// ---- tc_mca_std_lib/VISUs/PneumaticsVisu.TcVIS
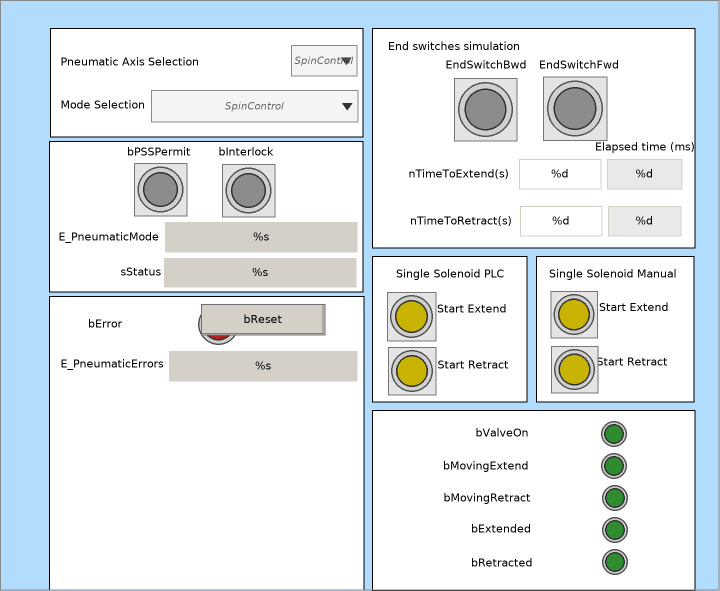
VISUALIZATION PneumaticsVisu  // 720x591
    Rectangle (50,28 313x109)
    Label (55,47 150x30), "Pneumatic Axis Selection"
    Rectangle (372,28 323x220)
    Label (379,30 150x33), "End switches simulation"
    Label (411,50 150x30), "EndSwitchBwd"
    SpinControl (291,45 66x31), variable: MAIN.hmiPneumaticAxisSelection
        p651134158: GVL_APP.nPNEUMATIC_AXIS_NUM
    Label (504,50 150x30), "EndSwitchFwd"
    Rectangle (49,296 315x294)
    Textfield (519,159 82x30), "%d", text variable: MAIN.afbPneumaticAxes[MAIN.hmiPneumaticAxisSelection].stPneumaticAxisStruct.stPneumaticAxisConfig.nTimeToExtend
        OnMouseClick: write MAIN.afbPneumaticAxes[MAIN.hmiPneumaticAxisSelection].stPneumaticAxisStruct.stPneumaticAxisConfig.nTimeToExtend via Default
    Label (384,159 150x30), "nTimeToExtend(s)"
    Label (386,206 150x30), "nTimeToRetract(s)"
    Label (28,90 150x30), "Mode Selection"
    Rectangle (49,141 314x151)
    Label (30,309 150x30), "bError"
    Lamp1 (126,301 185x47), variable: MAIN.afbPneumaticAxes[MAIN.hmiPneumaticAxisSelection].stPneumaticAxisStruct.stPneumaticAxisStatus.bError, style: Lamp-Lamp1-Red
    Label (37,349 150x30), "E_PneumaticErrors"
    Textfield (169,351 188x30), "%s", text variable: MAIN.afbPneumaticAxes[MAIN.hmiPneumaticAxisSelection].stPneumaticAxisStruct.ePneumaticAxisErrors, text list: 'languageSupport'
    Rectangle (372,256 155x146)
    Rectangle (536,256 158x146)
    Rectangle (372,410 323x181)
    Label (538,259 150x30), "Single Solenoid Manual"
    PushSwitchLed (549,291 50x47), variable: MAIN.afbPneumaticAxes[MAIN.hmiPneumaticAxisSelection].stPneumaticAxisStruct.stPneumaticAxisInputs.bOpenManual, behaviour: TOGGLE, style: Switch-PushSwitchLed-Yellow
    Label (592,293 84x29), "Start Extend"
    Label (557,347 150x30), "Start Retract"
    Label (375,259 150x30), "Single Solenoid PLC"
    PushSwitchLed (387,292 49x49), variable: MAIN.afbPneumaticAxes[MAIN.hmiPneumaticAxisSelection].stPneumaticAxisStruct.stPneumaticAxisControl.bExtend, behaviour: TOGGLE, style: Switch-PushSwitchLed-Yellow
    PushSwitchLed (388,347 48x48), variable: MAIN.afbPneumaticAxes[MAIN.hmiPneumaticAxisSelection].stPneumaticAxisStruct.stPneumaticAxisControl.bRetract, behaviour: TOGGLE, style: Switch-PushSwitchLed-Yellow
    Label (427,418 150x30), "bValveOn"
    Lamp1 (539,419 150x30), variable: MAIN.afbPneumaticAxes[MAIN.hmiPneumaticAxisSelection].stPneumaticAxisStruct.stPneumaticAxisOutputs.bValveOn, style: Lamp-Lamp1-Green
    Label (411,451 150x30), "bMovingExtend"
    Lamp1 (539,451 150x30), variable: MAIN.afbPneumaticAxes[MAIN.hmiPneumaticAxisSelection].stPneumaticAxisStruct.stPneumaticAxisStatus.bExtending, style: Lamp-Lamp1-Green
    Lamp1 (540,483 150x30), variable: MAIN.afbPneumaticAxes[MAIN.hmiPneumaticAxisSelection].stPneumaticAxisStruct.stPneumaticAxisStatus.bRetracting, style: Lamp-Lamp1-Green
    Lamp1 (540,515 150x30), variable: MAIN.afbPneumaticAxes[MAIN.hmiPneumaticAxisSelection].stPneumaticAxisStruct.stPneumaticAxisStatus.bExtended, style: Lamp-Lamp1-Green
    Lamp1 (540,547 150x30), variable: MAIN.afbPneumaticAxes[MAIN.hmiPneumaticAxisSelection].stPneumaticAxisStruct.stPneumaticAxisStatus.bRetracted, style: Lamp-Lamp1-Green
    Label (412,483 150x30), "bMovingRetract"
    Label (426,514 150x30), "bExtended"
    Label (397,294 150x30), "Start Extend"
    Label (398,350 150x30), "Start Retract"
    Label (427,548 150x30), "bRetracted"
    Button (201,304 124x31), "bReset"
        toggle MAIN.afbPneumaticAxes[MAIN.hmiPneumaticAxisSelection].stPneumaticAxisStruct.stPneumaticAxisControl.bReset
    PushSwitchLed (549,346 51x47), variable: MAIN.afbPneumaticAxes[MAIN.hmiPneumaticAxisSelection].stPneumaticAxisStruct.stPneumaticAxisInputs.bCloseManual, behaviour: TOGGLE, style: Switch-PushSwitchLed-Yellow
    Label (84,137 150x30), "bPSSPermit"
    Label (34,222 150x30), "E_PneumaticMode"
    Textfield (165,222 192x30), "%s", text variable: MAIN.afbPneumaticAxes[MAIN.hmiPneumaticAxisSelection].stPneumaticAxisStruct.ePneumaticAxisMode, text list: 'languageSupport'
    Textfield (164,258 192x29), "%s", text variable: MAIN.afbPneumaticAxes[MAIN.hmiPneumaticAxisSelection].stPneumaticAxisStruct.stPneumaticAxisStatus.sStatus, text list: 'languageSupport'
    Label (66,257 150x30), "sStatus"
    Textfield (520,206 82x30), "%d", text variable: MAIN.afbPneumaticAxes[MAIN.hmiPneumaticAxisSelection].stPneumaticAxisStruct.stPneumaticAxisConfig.nTimeToRetract
        OnMouseClick: write MAIN.afbPneumaticAxes[MAIN.hmiPneumaticAxisSelection].stPneumaticAxisStruct.stPneumaticAxisConfig.nTimeToRetract via Default
    Textfield (607,159 75x30), "%d", text variable: MAIN.afbPneumaticAxes[MAIN.hmiPneumaticAxisSelection].fbTimerExtend.ET
    Textfield (608,206 73x30), "%d", text variable: MAIN.afbPneumaticAxes[MAIN.hmiPneumaticAxisSelection].fbTimerRetract.ET
    SpinControl (151,90 207x32), variable: MAIN.afbPneumaticAxes[MAIN.hmiPneumaticAxisSelection].stPneumaticAxisStruct.ePneumaticAxisMode
    Label (570,132 150x30), "Elapsed time (ms)"
    PushSwitchLed (454,77 63x65), variable: MAIN.afbPneumaticAxes[MAIN.hmiPneumaticAxisSelection].stPneumaticAxisStruct.stPneumaticAxisInputs.bEndSwitchBwd, behaviour: TOGGLE, style: Switch-PushSwitchLed-Gray
    PushSwitchLed (543,76 64x65), variable: MAIN.afbPneumaticAxes[MAIN.hmiPneumaticAxisSelection].stPneumaticAxisStruct.stPneumaticAxisInputs.bEndSwitchFwd, behaviour: TOGGLE, style: Switch-PushSwitchLed-Gray
    PushSwitchLed (134,163 53x53), variable: MAIN.afbPneumaticAxes[MAIN.hmiPneumaticAxisSelection].stPneumaticAxisStruct.stPneumaticAxisInputs.bPSSPermit, behaviour: TOGGLE, style: Switch-PushSwitchLed-Gray
    PushSwitchLed (222,164 53x53), variable: MAIN.afbPneumaticAxes[MAIN.hmiPneumaticAxisSelection].stPneumaticAxisStruct.stPneumaticAxisControl.bInterlock, behaviour: TOGGLE, style: Switch-PushSwitchLed-Gray
    Label (171,137 150x30), "bInterlock"
END_VISUALIZATION

// ---- tc_mca_std_lib/VISUs_Org/languageSupport_1.TcTLO
TEXTLIST languageSupport_1
  axesAvailable = 'PLC Axes available: %d' | Test: 'Alt language'
  velocity = 'Velocity:'
  actposition = 'Actual Position:'
  enable = 'Enable Axis'
  enFW = 'Fwd Enable'
  enBW = 'Bwd Enable'
  axisSel = 'Axis Selected:'
  actVelocity = 'Actual Velocity:'
  errID = 'Error ID:'
  bEnabled = 'Axis Enabled'
  bCommandAborted = 'Command Aborted'
  bBusy = 'Busy'
  bDone = 'Command Done'
  bResetDone = 'Reset Complete'
  bHomed = 'Calibrated'
  bFwEnabled = 'Fwd movement enabled'
  bBwEnabled = 'Bwd movement enabled'
  bError = 'Error'
  fVelocity = 'Target Velocity:'
  fAcceleration = 'Target Accel.:'
  fDeceleration = 'Target Decel.:'
  fPosition = 'Target Position:'
  moveAbsolute = 'Absolute position move'
  toggle = 'Toggle'
  moveVelocity = 'Constant velocity move'
  bExecute = 'Motion function executed'
  moveRelative = 'Relative position move'
  moveModulo = 'Modulo position move'
  reset = 'Reset axis'
  stop = 'Stop motion'
  jogBw = 'Jog Backward'
  jogFw = 'Jog Forward'
  bGeared = 'In Gear'
  masterGear = 'Master Axis'
  gearRatio = 'Gear Ratio'
  gearIn = 'Gear In'
  gearOut = 'Gear Out'
  eHomeToLimit_Bwd = 'Bwd Limit'
  eHomeToLimit_Fwd = 'Fwd Limit'
  eHomeToRef_Bwd = 'Home Switch Bwd '
  eHomeToRef_Fwd = 'Home Switch Fwd '
  eHomeToEncPulse_Bwd = 'Enc Pulse Bwd '
  eHomeToEncPulse_Fwd = 'Enc Pulse Fwd'
  eHomeToEncPulse_viaBwdLimit = 'Enc Pulse via Bwd Limit'
  eHomeToEncPulse_viaFwdLimit = 'Enc Pulse via Fwd Limit'
  eHomeToBlock_Bwd = 'Home To Block Bwd Lag Based'
  eHomeToBlock_Fwd = 'Home To Block Fwd Lag Based'
  eHomeDirect = 'Home Direct'
  fHomePosition = 'Set Pos after Homing'
  fHomeFinishDistance = 'Relative Move after Homing'
  halt = 'Halt Motion'
  bInterlockBwd = 'Interlock Bwd'
  bInterlockFwd = 'Interlock Fwd'
  Home = 'HOME'
  eWriteParameter = 'Write Parameter'
  eReadParameter = 'Read Parameter'
  fWriteAxisParameter = 'Parameter to write'
  fReadAxisParameter = 'Parameter'
  bLocalMode = 'Local Mode'
  bInVelocity = 'Target Velocity reached'
   = ''
END_TEXTLIST

// ---- tc_mca_std_lib/VISUs_Org/MainVisu_1.TcVIS
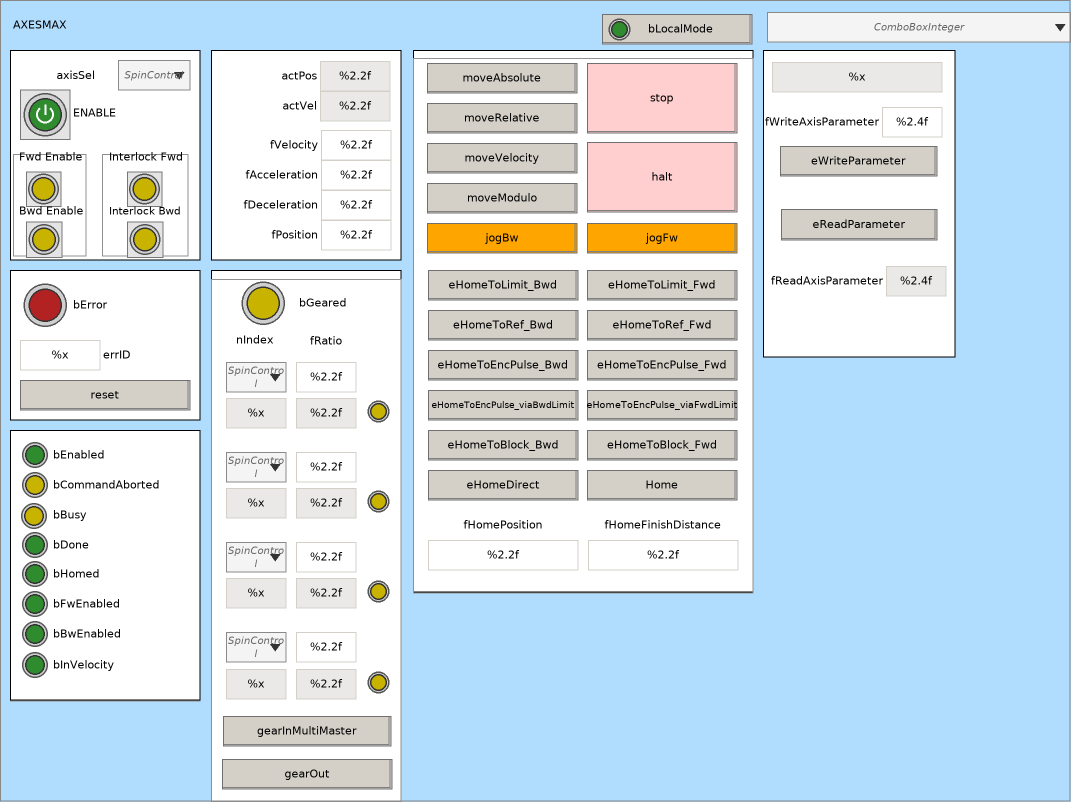
VISUALIZATION MainVisu_1  // 1071x802
    Rectangle (413,50 340x542)
    GroupBox (413,50 340x543)
        Button (174,92 150x70), "halt", pressed state: GVL.astAxes[Main.hmiAxisSelection].stControl.bHalt, input disabled if: GVL.astAxes[MAIN.hmiAxisSelection].stStatus.bGeared, text list: "languageSupport", text index: "halt"
            toggle GVL.astAxes[Main.hmiAxisSelection].stControl.bHalt
        Button (174,420 150x30), "Home", input disabled if: GVL.astAxes[MAIN.hmiAxisSelection].stStatus.bGeared, text list: 'languageSupport', text index: "Home"
            OnMouseClick: execute { GVL.astAxes[Main.hmiAxisSelection].stControl.eCommand:=E_MotionFunctions.eHome; GVL.astAxes[Main.hmiAxisSelection].stControl.bExecute:=TRUE; }
        Button (15,380 150x30), "eHomeToBlock_Bwd", input disabled if: GVL.astAxes[MAIN.hmiAxisSelection].stStatus.bGeared, text list: 'languageSupport', text index: "eHomeToBlock_Bwd"
            OnMouseClick: execute {
                GVL.astAxes[Main.hmiAxisSelection].stControl.eCommand:=E_MotionFunctions.eHome;
                GVL.astAxes[Main.hmiAxisSelection].stConfig.eHomeSeq:=E_HomingRoutines.eHomeToBlock_Bwd;
                GVL.astAxes[Main.hmiAxisSelection].stControl.bExecute:=TRUE;
            }
    Rectangle (211,270 190x531)
    GroupBox (211,271 190x531)
        SpinControl (15,91 60x30), variable: GVL.astAxes[MAIN.hmiAxisSelection].stConfig.astMultiMasterAxis[1].nIndex
            p651134158: GVL_APP.nAXIS_NUM
        Textfield (85,91 60x30), "%2.2f", text variable: GVL.astAxes[MAIN.hmiAxisSelection].stConfig.astMultiMasterAxis[1].fRatio
            OnMouseClick: write the text variable via Default
        Textfield (80,55 70x30), "fRatio", text list: "languageSupport", text index: "gearRatio"
        Button (12,445 168x30), "gearInMultiMaster", text list: "languageSupport", text index: "gearIn"
            OnMouseClick: execute { GVL.astAxes[Main.hmiAxisSelection].stControl.eCommand:=E_MotionFunctions.eGearInMultiMaster; GVL.astAxes[Main.hmiAxisSelection].stControl.bExecute:=TRUE; }
        SpinControl (15,181 60x30), variable: GVL.astAxes[MAIN.hmiAxisSelection].stConfig.astMultiMasterAxis[2].nIndex
            p651134158: GVL_APP.nAXIS_NUM
        SpinControl (15,271 60x30), variable: GVL.astAxes[MAIN.hmiAxisSelection].stConfig.astMultiMasterAxis[3].nIndex
            p651134158: GVL_APP.nAXIS_NUM
        SpinControl (15,361 60x30), variable: GVL.astAxes[MAIN.hmiAxisSelection].stConfig.astMultiMasterAxis[4].nIndex
            p651134158: GVL_APP.nAXIS_NUM
        Textfield (85,181 60x30), "%2.2f", text variable: GVL.astAxes[MAIN.hmiAxisSelection].stConfig.astMultiMasterAxis[2].fRatio
            OnMouseClick: write the text variable via Default
        Textfield (85,271 60x30), "%2.2f", text variable: GVL.astAxes[MAIN.hmiAxisSelection].stConfig.astMultiMasterAxis[3].fRatio
            OnMouseClick: write the text variable via Default
        Textfield (85,361 60x30), "%2.2f", text variable: GVL.astAxes[MAIN.hmiAxisSelection].stConfig.astMultiMasterAxis[4].fRatio
            OnMouseClick: write the text variable via Default
        Button (11,488 170x30), "gearOut", text list: "languageSupport", text index: "gearOut"
            OnMouseClick: execute { GVL.astAxes[Main.hmiAxisSelection].stControl.eCommand:=E_MotionFunctions.eGearOut; GVL.astAxes[Main.hmiAxisSelection].stControl.bExecute:=TRUE; }
        Textfield (9,54 70x30), "nIndex", text list: "languageSupport", text index: "masterGear"
        Textfield (85,127 60x30), "%2.2f", text variable: GVL.astAxes[MAIN.hmiAxisSelection].Axis.PlcToNc.GearRatio1
        Textfield (15,127 60x30), "%x", text variable: GVL.astAxes[MAIN.hmiAxisSelection].stConfig.astMultiMasterAxisLatched[1].nIndex
        Textfield (85,217 60x30), "%2.2f", text variable: GVL.astAxes[MAIN.hmiAxisSelection].Axis.PlcToNc.GearRatio2
        Textfield (15,217 60x30), "%x", text variable: GVL.astAxes[MAIN.hmiAxisSelection].stConfig.astMultiMasterAxisLatched[2].nIndex
        Textfield (85,307 60x30), "%2.2f", text variable: GVL.astAxes[MAIN.hmiAxisSelection].Axis.PlcToNc.GearRatio3
        Textfield (15,307 60x30), "%x", text variable: GVL.astAxes[MAIN.hmiAxisSelection].stConfig.astMultiMasterAxisLatched[3].nIndex
        Textfield (85,398 60x30), "%2.2f", text variable: GVL.astAxes[MAIN.hmiAxisSelection].Axis.PlcToNc.GearRatio4
        Textfield (15,398 60x30), "%x", text variable: GVL.astAxes[MAIN.hmiAxisSelection].stConfig.astMultiMasterAxisLatched[4].nIndex
        Lamp1 (155,399 25x25), variable: GVL.astAxes[MAIN.hmiAxisSelection].stStatus.bCoupledGear4, style: Lamp-Lamp1-Yellow
        Lamp1 (155,308 25x25), variable: GVL.astAxes[MAIN.hmiAxisSelection].stStatus.bCoupledGear3, style: Lamp-Lamp1-Yellow
        Lamp1 (155,218 25x25), variable: GVL.astAxes[MAIN.hmiAxisSelection].stStatus.bCoupledGear2, style: Lamp-Lamp1-Yellow
        Lamp1 (155,128 25x25), variable: GVL.astAxes[MAIN.hmiAxisSelection].stStatus.bCoupledGear1, style: Lamp-Lamp1-Yellow
        Lamp1 (27,7 50x50), variable: GVL.astAxes[MAIN.hmiAxisSelection].stStatus.bGeared, style: Lamp-Lamp1-Yellow
    GroupBox (10,50 190x210)
        Rectangle (0,0 190x210)
        GroupBox (3,96 73x110)
        GroupBox (92,96 86x110)
        Textfield (60,50 92x26), "ENABLE", text list: 'languageSupport', text index: "enable"
        PushSwitchLed (16,118 35x42), variable: GVL.astAxes[MAIN.hmiAxisSelection].stInputs.bLimitFwd, behaviour: TOGGLE, style: Switch-PushSwitchLed-Yellow
        PushSwitchLed (16,170 36x39), variable: GVL.astAxes[MAIN.hmiAxisSelection].stInputs.bLimitBwd, behaviour: TOGGLE, style: Switch-PushSwitchLed-Yellow
        SpinControl (108,10 72x30), variable: MAIN.hmiAxisSelection
            p651134158: GVL_APP.nAXIS_NUM
        Textfield (23,13 86x25), "axisSel", text variable: GVL_APP.nAXIS_NUM, text list: "languageSupport", text index: "axisSel"
        PowerSwitch (10,38 50x53), variable: GVL.astAxes[MAIN.hmiAxisSelection].stControl.bEnable, behaviour: TOGGLE, style: Switch-PowerSwitch-Green
        PushSwitchLed (117,118 35x42), variable: GVL.astAxes[MAIN.hmiAxisSelection].stControl.bInterlockFwd, behaviour: TOGGLE, style: Switch-PushSwitchLed-Yellow
        PushSwitchLed (117,170 36x39), variable: GVL.astAxes[MAIN.hmiAxisSelection].stControl.bInterlockBwd, behaviour: TOGGLE, style: Switch-PushSwitchLed-Yellow
        Textfield (6,94 76x26), "Fwd Enable", text list: 'languageSupport', text index: "enFW"
        Textfield (6,148 76x26), "Bwd Enable", text list: 'languageSupport', text index: "enBW"
        Textfield (96,94 76x26), "Interlock Fwd", text list: 'languageSupport', text index: "bAxisInterlockFwd"
        Textfield (96,148 76x26), "Interlock Bwd", text list: 'languageSupport', text index: "bAxisInterlockBwd"
    Textfield (10,10 231x30), "AXESMAX", text variable: GVL_APP.nAXIS_NUM, text list: "languageSupport", text index: "axesAvailable"
    Button (427,63 150x30), "moveAbsolute", text list: "languageSupport", text index: "moveAbsolute"
        OnMouseClick: execute { GVL.astAxes[MAIN.hmiAxisSelection].stControl.eCommand:=E_MotionFunctions.eMoveAbsolute; GVL.astAxes[MAIN.hmiAxisSelection].stControl.bExecute:=TRUE; }
    Button (427,143 150x30), "moveVelocity", input disabled if: GVL.astAxes[MAIN.hmiAxisSelection].stStatus.bGeared, text list: "languageSupport", text index: "moveVelocity"
        OnMouseClick: execute { GVL.astAxes[Main.hmiAxisSelection].stControl.eCommand:=E_MotionFunctions.eMoveVelocity; GVL.astAxes[Main.hmiAxisSelection].stControl.bExecute:=TRUE; }
    Button (427,103 150x30), "moveRelative", input disabled if: GVL.astAxes[MAIN.hmiAxisSelection].stStatus.bGeared, text list: "languageSupport", text index: "moveRelative"
        OnMouseClick: execute { GVL.astAxes[Main.hmiAxisSelection].stControl.eCommand:=E_MotionFunctions.eMoveRelative; GVL.astAxes[Main.hmiAxisSelection].stControl.bExecute:=TRUE; }
    Button (427,183 150x30), "moveModulo", input disabled if: GVL.astAxes[MAIN.hmiAxisSelection].stStatus.bGeared, text list: "languageSupport", text index: "moveModulo"
        OnMouseClick: execute { GVL.astAxes[Main.hmiAxisSelection].stControl.eCommand:=E_MotionFunctions.eMoveModulo; GVL.astAxes[Main.hmiAxisSelection].stControl.bExecute:=TRUE; }
    Button (587,63 150x70), "stop", pressed state: GVL.astAxes[Main.hmiAxisSelection].stControl.bStop, input disabled if: GVL.astAxes[MAIN.hmiAxisSelection].stStatus.bGeared, text list: "languageSupport", text index: "stop"
        toggle GVL.astAxes[Main.hmiAxisSelection].stControl.bStop
    Button (427,223 150x30), "jogBw", text list: "languageSupport", text index: "jogBw"
        OnMouseClick: execute {  }
        OnMouseDown: execute {
            GVL.astAxes[Main.hmiAxisSelection].stControl.eCommand:=E_MotionFunctions.eMoveVelocity;
            GVL.astAxes[Main.hmiAxisSelection].stControl.fVelocity:=-ABS(GVL.astAxes[Main.hmiAxisSelection].stControl.fJogVelocity)
            GVL.astAxes[Main.hmiAxisSelection].stControl.bExecute:= TRUE;
        }
        OnMouseUp: execute { GVL.astAxes[Main.hmiAxisSelection].stControl.bHalt:= TRUE; }
    Button (587,223 150x30), "jogFw", text list: "languageSupport", text index: "jogFw"
        OnMouseClick: execute {  }
        OnMouseDown: execute {
            GVL.astAxes[Main.hmiAxisSelection].stControl.eCommand:=E_MotionFunctions.eMoveVelocity;
            GVL.astAxes[Main.hmiAxisSelection].stControl.fVelocity:=ABS(GVL.astAxes[Main.hmiAxisSelection].stControl.fJogVelocity)
            GVL.astAxes[Main.hmiAxisSelection].stControl.bExecute:= TRUE;
        }
        OnMouseUp: execute { GVL.astAxes[Main.hmiAxisSelection].stControl.bHalt:= TRUE; }
    GroupBox (10,270 190x150)
        Rectangle (0,0 190x150)
        Textfield (90,70 90x30), "errID", text list: "languageSupport", text index: "errID"
        Textfield (10,70 80x30), "%x", text variable: GVL.astAxes[MAIN.hmiAxisSelection].stStatus.nErrorID
        Lamp1 (10,10 50x50), variable: GVL.astAxes[MAIN.hmiAxisSelection].stStatus.bError, style: Lamp-Lamp1-Red
        Textfield (60,20 120x30), "bError", text list: "languageSupport", text index: "bError"
        Button (10,110 170x30), "reset", pressed state: GVL.astAxes[Main.hmiAxisSelection].stControl.bReset, text list: "languageSupport", text index: "reset"
            OnMouseClick: toggle GVL.astAxes[Main.hmiAxisSelection].stControl.bReset
    GroupBox (10,430 190x271)
        Rectangle (0,0 190x270)
        Lamp1 (10,10 30x30), variable: GVL.astAxes[MAIN.hmiAxisSelection].stStatus.bEnabled, style: Lamp-Lamp1-Green
        Textfield (40,10 140x30), "bEnabled", text list: "languageSupport", text index: "bEnabled"
        Lamp1 (10,40 30x30), variable: GVL.astAxes[MAIN.hmiAxisSelection].stStatus.bCommandAborted, style: Lamp-Lamp1-Yellow
        Textfield (40,40 140x30), "bCommandAborted", text list: "languageSupport", text index: "bWarning"
        Textfield (40,70 140x30), "bBusy", text list: "languageSupport", text index: "bBusy"
        Lamp1 (10,100 30x30), variable: GVL.astAxes[MAIN.hmiAxisSelection].stStatus.bDone, style: Lamp-Lamp1-Green
        Textfield (40,100 140x30), "bDone", text list: 'languageSupport', text index: "bDone"
        Lamp1 (10,129 30x30), variable: GVL.astAxes[MAIN.hmiAxisSelection].stStatus.bHomed, style: Lamp-Lamp1-Green
        Textfield (40,129 140x30), "bHomed", text list: "languageSupport", text index: "bHomed"
        Lamp1 (10,159 30x30), variable: GVL.astAxes[MAIN.hmiAxisSelection].stStatus.bFwEnabled AND NOT GVL.astAxes[MAIN.hmiAxisSelection].stStatus.bInterlockedFwd, style: Lamp-Lamp1-Green
        Lamp1 (10,189 30x30), variable: GVL.astAxes[MAIN.hmiAxisSelection].stStatus.bBwEnabled AND NOT GVL.astAxes[MAIN.hmiAxisSelection].stStatus.bInterlockedBwd, style: Lamp-Lamp1-Green
        Textfield (40,159 140x30), "bFwEnabled", text list: "languageSupport", text index: "bFwEnabled"
        Textfield (40,189 140x30), "bBwEnabled", text list: "languageSupport", text index: "bBwEnabled"
        Lamp1 (9,71 30x30), variable: GVL.astAxes[MAIN.hmiAxisSelection].stStatus.bBusy, style: Lamp-Lamp1-Yellow
        Lamp1 (10,220 30x30), variable: GVL.astAxes[MAIN.hmiAxisSelection].stStatus.bInVelocity, style: Lamp-Lamp1-Green
    GroupBox (211,50 190x210)
        Rectangle (0,0 190x210)
        Textfield (10,80 100x30), "fVelocity", text list: "languageSupport", text index: "fVelocity"
        Textfield (110,80 70x30), "%2.2f", text variable: GVL.astAxes[MAIN.hmiAxisSelection].stControl.fVelocity
            OnMouseClick: write the text variable via Default
        Textfield (10,110 100x30), "fAcceleration", text list: "languageSupport", text index: "fAcceleration"
        Textfield (110,110 70x30), "%2.2f", text variable: GVL.astAxes[MAIN.hmiAxisSelection].stControl.fAcceleration
            OnMouseClick: write the text variable via Default
        Textfield (10,140 100x30), "fDeceleration", text list: "languageSupport", text index: "fDeceleration"
        Textfield (110,140 70x30), "%2.2f", text variable: GVL.astAxes[MAIN.hmiAxisSelection].stControl.fDeceleration
            OnMouseClick: write the text variable via Default
        Textfield (10,170 100x30), "fPosition", text list: "languageSupport", text index: "fPosition"
        Textfield (110,170 70x30), "%2.2f", text variable: GVL.astAxes[MAIN.hmiAxisSelection].stControl.fPosition
            OnMouseClick: write the text variable via Default
        Textfield (109,11 70x30), "%2.2f", text variable: GVL.astAxes[MAIN.hmiAxisSelection].stStatus.fActPosition
        Textfield (9,11 100x30), "actPos", text list: "languageSupport", text index: "actposition"
        Textfield (9,41 100x30), "actVel", text list: "languageSupport", text index: "actVelocity"
        Textfield (109,41 70x30), "%2.2f", text variable: GVL.astAxes[MAIN.hmiAxisSelection].stStatus.fActVelocity
    Button (428,310 150x30), "eHomeToRef_Bwd", input disabled if: GVL.astAxes[MAIN.hmiAxisSelection].stStatus.bGeared, text list: 'languageSupport', text index: "eHomeToRef_Bwd"
        OnMouseClick: execute {
            GVL.astAxes[Main.hmiAxisSelection].stControl.eCommand:=E_MotionFunctions.eHome;
            GVL.astAxes[Main.hmiAxisSelection].stConfig.eHomeSeq:=E_HomingRoutines.eHomeToRef_Bwd;
            GVL.astAxes[Main.hmiAxisSelection].stControl.bExecute:=TRUE;
        }
    Button (587,310 150x30), "eHomeToRef_Fwd", input disabled if: GVL.astAxes[MAIN.hmiAxisSelection].stStatus.bGeared, text list: "languageSupport", text index: "eHomeToRef_Fwd"
        OnMouseClick: execute {
            GVL.astAxes[Main.hmiAxisSelection].stControl.eCommand:=E_MotionFunctions.eHome;
            GVL.astAxes[Main.hmiAxisSelection].stConfig.eHomeSeq:=E_HomingRoutines.eHomeToRef_Fwd;
            GVL.astAxes[Main.hmiAxisSelection].stControl.bExecute:=TRUE;
        }
    Textfield (296,288 93x30), "bGeared", text list: "languageSupport", text index: "bGeared"
    Button (428,350 150x30), "eHomeToEncPulse_Bwd", input disabled if: GVL.astAxes[MAIN.hmiAxisSelection].stStatus.bGeared, text list: 'languageSupport', text index: "eHomeToEncPulse_Bwd"
        OnMouseClick: execute {
            GVL.astAxes[Main.hmiAxisSelection].stControl.eCommand:=E_MotionFunctions.eHome;
            GVL.astAxes[Main.hmiAxisSelection].stConfig.eHomeSeq:=E_HomingRoutines.eHomeToEncPulse_Bwd;
            GVL.astAxes[Main.hmiAxisSelection].stControl.bExecute:=TRUE;
        }
    Button (587,350 150x30), "eHomeToEncPulse_Fwd", input disabled if: GVL.astAxes[MAIN.hmiAxisSelection].stStatus.bGeared, text list: "languageSupport", text index: "eHomeToEncPulse_Fwd"
        OnMouseClick: execute {
            GVL.astAxes[Main.hmiAxisSelection].stControl.eCommand:=E_MotionFunctions.eHome;
            GVL.astAxes[Main.hmiAxisSelection].stConfig.eHomeSeq:=E_HomingRoutines.eHomeToEncPulse_Fwd;
            GVL.astAxes[Main.hmiAxisSelection].stControl.bExecute:=TRUE;
        }
    Button (428,470 150x30), "eHomeDirect", input disabled if: GVL.astAxes[MAIN.hmiAxisSelection].stStatus.bGeared, text list: 'languageSupport', text index: "eHomeDirect"
        OnMouseClick: execute {
            GVL.astAxes[Main.hmiAxisSelection].stControl.eCommand:=E_MotionFunctions.eHome;
            GVL.astAxes[Main.hmiAxisSelection].stConfig.eHomeSeq:=E_HomingRoutines.eHomeDirect;
            GVL.astAxes[Main.hmiAxisSelection].stControl.bExecute:=TRUE;
        }
    Button (428,270 150x30), "eHomeToLimit_Bwd", input disabled if: GVL.astAxes[MAIN.hmiAxisSelection].stStatus.bGeared, text list: 'languageSupport', text index: "eHomeToLimit_Bwd"
        OnMouseClick: execute {
            GVL.astAxes[Main.hmiAxisSelection].stControl.eCommand:=E_MotionFunctions.eHome;
            GVL.astAxes[Main.hmiAxisSelection].stConfig.eHomeSeq:=E_HomingRoutines.eHomeToLimit_Bwd;
            GVL.astAxes[Main.hmiAxisSelection].stControl.bExecute:=TRUE;
        }
    Button (587,270 150x30), "eHomeToLimit_Fwd", input disabled if: GVL.astAxes[MAIN.hmiAxisSelection].stStatus.bGeared, text list: "languageSupport", text index: "eHomeToLimit_Fwd"
        OnMouseClick: execute {
            GVL.astAxes[Main.hmiAxisSelection].stControl.eCommand:=E_MotionFunctions.eHome;
            GVL.astAxes[Main.hmiAxisSelection].stConfig.eHomeSeq:=E_HomingRoutines.eHomeToLimit_Fwd;
            GVL.astAxes[Main.hmiAxisSelection].stControl.bExecute:=TRUE;
        }
    Textfield (428,540 150x30), "%2.2f", text variable: GVL.astAxes[MAIN.hmiAxisSelection].stConfig.fHomePosition
        OnMouseClick: write the text variable via Default
    Button (428,390 150x30), "eHomeToEncPulse_viaBwdLimit", input disabled if: GVL.astAxes[MAIN.hmiAxisSelection].stStatus.bGeared, text list: 'languageSupport', text index: "eHomeToEncPulse_viaBwdLimit"
        OnMouseClick: execute {
            GVL.astAxes[Main.hmiAxisSelection].stControl.eCommand:=E_MotionFunctions.eHome;
            GVL.astAxes[Main.hmiAxisSelection].stConfig.eHomeSeq:=E_HomingRoutines.eHomeToEncPulse_viaBwdLimit;
            GVL.astAxes[Main.hmiAxisSelection].stControl.bExecute:=TRUE;
        }
    Button (587,390 150x30), "eHomeToEncPulse_viaFwdLimit", input disabled if: GVL.astAxes[MAIN.hmiAxisSelection].stStatus.bGeared, text list: "languageSupport", text index: "eHomeToEncPulse_viaFwdLimit"
        OnMouseClick: execute {
            GVL.astAxes[Main.hmiAxisSelection].stControl.eCommand:=E_MotionFunctions.eHome;
            GVL.astAxes[Main.hmiAxisSelection].stConfig.eHomeSeq:=E_HomingRoutines.eHomeToEncPulse_viaFwdLimit;
            GVL.astAxes[Main.hmiAxisSelection].stControl.bExecute:=TRUE;
        }
    Textfield (588,540 150x30), "%2.2f", text variable: GVL.astAxes[MAIN.hmiAxisSelection].stConfig.fHomeFinishDistance
        OnMouseClick: write the text variable via Default
    Textfield (428,510 150x30), "fHomePosition", text list: "languageSupport", text index: "fHomePosition"
    Textfield (588,510 150x30), "fHomeFinishDistance", text list: "languageSupport", text index: "fHomeFinishDistance"
    Group (602,14 150x30)
        Button (0,0 150x30), "bLocalMode", text list: 'languageSupport', text index: bLocalMode
            OnMouseClick: toggle bLocalMode
        Lamp1 (5,3 25x25), variable: bLocalMode, style: Lamp-Lamp1-Green
    Rectangle (763,50 192x307)
    Button (780,146 157x30), "eWriteParameter", input disabled if: GVL.astAxes[MAIN.hmiAxisSelection].stStatus.bGeared, text list: "languageSupport", text index: "eWriteParameter"
        OnMouseClick: execute { GVL.astAxes[MAIN.hmiAxisSelection].stControl.eCommand:=E_MotionFunctions.eWriteParameter; GVL.astAxes[MAIN.hmiAxisSelection].stControl.bExecute:=TRUE; }
    Textfield (772,62 170x30), "%x", text variable: astAxes[MAIN.hmiAxisSelection].stConfig.eAxisParameters
        OnMouseClick: write GVL.astAxes[MAIN.hmiAxisSelection].stConfig.eAxisParameters via Default
    Textfield (762,107 120x30), "fWriteAxisParameter", text list: "languageSupport", text index: "fWriteAxisParameter"
    Textfield (882,107 60x30), "%2.4f", text variable: astAxes[MAIN.hmiAxisSelection].stConfig.fWriteAxisParameter
        OnMouseClick: write GVL.astAxes[MAIN.hmiAxisSelection].stConfig.fWriteAxisParameter via Default
    Textfield (886,266 60x30), "%2.4f", text variable: astAxes[MAIN.hmiAxisSelection].stConfig.fReadAxisParameter
        OnMouseClick: write GVL.astAxes[MAIN.hmiAxisSelection].stConfig.fReadAxisParameter via Default
    Textfield (766,266 120x30), "fReadAxisParameter", text list: "languageSupport", text index: "fReadAxisParameter"
    Button (781,209 156x31), "eReadParameter", input disabled if: GVL.astAxes[MAIN.hmiAxisSelection].stStatus.bGeared, text list: 'languageSupport', text index: "eReadParameter"
        OnMouseClick: execute { GVL.astAxes[MAIN.hmiAxisSelection].stControl.eCommand:=E_MotionFunctions.eReadParameter; GVL.astAxes[MAIN.hmiAxisSelection].stControl.bExecute:=TRUE; }
    ComboBoxInteger (767,12 304x30), variable: GVL.astAxes[MAIN.hmiAxisSelection].stConfig.eAxisParameters, text list: 'ParameterTextList'
    Textfield (50,650 140x30), "bInVelocity", text list: 'languageSupport', text index: "bInVelocity"
    Button (587,430 150x30), "eHomeToBlock_Fwd", input disabled if: GVL.astAxes[MAIN.hmiAxisSelection].stStatus.bGeared, text list: "languageSupport", text index: "eHomeToBlock_Fwd"
        OnMouseClick: execute {
            GVL.astAxes[Main.hmiAxisSelection].stControl.eCommand:=E_MotionFunctions.eHome;
            GVL.astAxes[Main.hmiAxisSelection].stConfig.eHomeSeq:=E_HomingRoutines.eHomeToBlock_Fwd;
            GVL.astAxes[Main.hmiAxisSelection].stControl.bExecute:=TRUE;
        }
END_VISUALIZATION

// ---- tc_mca_std_lib/VISUs_Org/ParameterTextList_1.TcTLO
TEXTLIST ParameterTextList_1
  1 = 'CommandedPosition'
  2 = 'SWLimitForward'
  3 = 'SWLimitBackward'
  4 = 'EnableLimitForward'
  5 = 'EnableLimitBackward'
  6 = 'EnablePositionLagMonitoring'
  7 = 'MaxPositionLag'
  8 = 'AxisMaxVelocity'
  10 = 'ActualVelocity'
  11 = 'CommandedVelocity'
  12 = 'AxisDefaultAcceleration'
  14 = 'AxisDefaultDeceleration'
  16 = 'AxisDefaultJerk'
  1000 = 'AxisId'
  1001 = 'AxisManualVelocitySlow'
  1002 = 'AxisManualVelocityFast'
  1009 = 'AxisRapidTraverseVelocity'
  1012 = 'AxisVelocityToCam'
  1013 = 'AxisVelocityFromCam'
  1014 = 'AxisJogIncrementForward'
  1015 = 'AxisJogIncrementBackward'
  1022 = 'MaxPositionLagFilterTime'
  1023 = 'AxisEnPositionRangeMonitoring'
  1024 = 'AxisPositionRangeWindow'
  1025 = 'AxisEnTargetPositionMonitoring'
  1026 = 'AxisTargetPositionWindow'
  1027 = 'AxisTargetPositionMonitoringTime'
  1028 = 'AxisEnInTargetTimeout'
  1029 = 'AxisInTargetTimeout'
  1030 = 'AxisEnMotionMonitoring'
  1031 = 'AxisMotionMonitoringWindow'
  1032 = 'AxisMotionMonitoringTime'
  1033 = 'AxisDelayTimeVeloPosition'
  1034 = 'AxisEnLoopingDistance'
  1035 = 'AxisLoopingDistance'
  1038 = 'AxisEnDataPersistence'
  1039 = 'AxisRefVeloOnRefOutput'
  1040 = 'AxisOverrideType'
  1042 = 'AxisEncoderOffset'
  1043 = 'AxisEncoderDirectionInverse'
  1044 = 'AxisEncoderMask'
  1045 = 'AxisEncoderModuloValue'
  1046 = 'AxisModuloToleranceWindow'
  1047 = 'AxisEnablePosCorrection'
  1048 = 'AxisPosCorrectionFilterTime'
  1049 = 'AxisUnitInterpretation'
  1050 = 'AxisMotorDirectionInverse'
  1051 = 'AxisCycleTime'
  1052 = 'AxisFastStopSignalType'
  1053 = 'AxisFastAcc'
  1054 = 'AxisFastDec'
  1055 = 'AxisFastJerk'
  1056 = 'AxisEncoderScalingNumerator'
  1057 = 'AxisEncoderScalingDenominator'
  1058 = 'AxisMaximumAcceleration'
  1059 = 'AxisMaximumDeceleration'
  1060 = 'AxisVeloJumpFactor'
  1061 = 'AxisToleranceBallAuxAxis'
  1062 = 'AxisMaxPositionDeviationAuxAxis'
  1063 = 'AxisErrorPropagationMode'
  1064 = 'AxisErrorPropagationDelay'
  1065 = 'AxisCoupleSlaveToActualValues'
  1066 = 'AxisAllowMotionCmdToSlaveAxis'
  1067 = 'AxisAllowMotionCmdToExtSetAxis'
  1068 = 'AxisEncoderSubMask'
  1069 = 'AxisEncoderReferenceSystem'
  1070 = 'AxisEncoderPositionFilterPT1'
  1071 = 'AxisEncoderVelocityFilterPT1'
  1072 = 'AxisEncoderAccelerationFilterPT1'
  1073 = 'AxisEncoderMode'
  1074 = 'AxisEncoderHomingInvDirCamSearch'
  1075 = 'AxisEncoderHomingInvDirSyncSearch'
  1076 = 'AxisEncoderHomingCalibValue'
  1077 = 'AxisEncoderReferenceMode'
  1078 = 'AxisRefVeloOutputRatio'
  1079 = 'AxisDrivePositionOutputScaling'
  1080 = 'AxisDriveVelocityOutputScaling'
  1081 = 'AxisDriveVelocityOutputDelay'
  1082 = 'AxisDriveMinOutputLimitation'
  1083 = 'AxisDriveMaxOutputLimitation'
  1084 = 'AxisTorqueInputScaling'
  1085 = 'AxisTorqueInputFilterPT1'
  1086 = 'AxisTorqueDerivationInputFilterPT1'
  1087 = 'AxisTorqueOutputScaling'
  1088 = 'AxisTorqueOutputDelay'
  1089 = 'AxisAccelerationOutputScaling'
  1090 = 'AxisAccelerationOutputDelay'
  1091 = 'AxisDrivePositionOutputSmoothFilterType'
  1092 = 'AxisDrivePositionOutputSmoothFilterTime'
  1093 = 'AxisDrivePositionOutputSmoothFilterOrder'
  1094 = 'AxisDriveMode'
  1095 = 'AxisDriftCompensationOffset'
  1096 = 'AxisPositionControlKv'
  1097 = 'AxisCtrlVelocityPreCtrlWeight'
  1098 = 'AxisControllerMode'
  1099 = 'AxisCtrlAutoOffset'
  1100 = 'AxisCtrlAutoOffsetTimer'
  1101 = 'AxisCtrlAutoOffsetLimit'
  1102 = 'AxisSlaveCouplingControlKcp'
  1103 = 'AxisCtrlOutputLimit'
  2000 = 'AxisTargetPosition'
  2001 = 'AxisRemainingTimeToGo'
  2002 = 'AxisRemainingDistanceToGo'
  3000 = 'AxisGearRatio'
  4000 = 'NcSafCycleTime'
  4001 = 'NcSvbCycleTime'
   = ''
END_TEXTLIST

// ---- tc_mca_std_lib/VISUs_Org/PneumaticsVisu_1.TcVIS
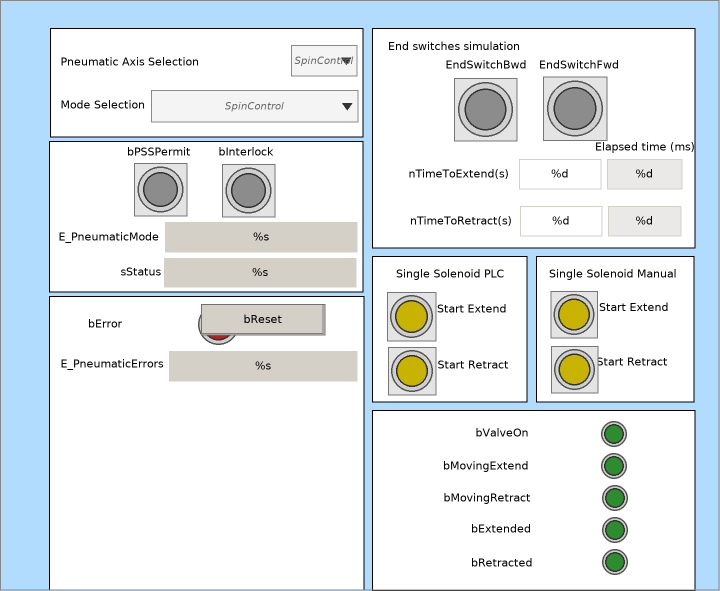
VISUALIZATION PneumaticsVisu_1  // 720x591
    Rectangle (50,28 313x109)
    Label (55,47 150x30), "Pneumatic Axis Selection"
    Rectangle (372,28 323x220)
    Label (379,30 150x33), "End switches simulation"
    Label (411,50 150x30), "EndSwitchBwd"
    SpinControl (291,45 66x31), variable: MAIN.hmiPneumaticAxisSelection
        p651134158: GVL_APP.nPNEUMATIC_AXIS_NUM
    Label (504,50 150x30), "EndSwitchFwd"
    Rectangle (49,296 315x294)
    Textfield (519,159 82x30), "%d", text variable: MAIN.afbPneumaticAxes[MAIN.hmiPneumaticAxisSelection].stPneumaticAxisStruct.stPneumaticAxisConfig.nTimeToExtend
        OnMouseClick: write MAIN.afbPneumaticAxes[MAIN.hmiPneumaticAxisSelection].stPneumaticAxisStruct.stPneumaticAxisConfig.nTimeToExtend via Default
    Label (384,159 150x30), "nTimeToExtend(s)"
    Label (386,206 150x30), "nTimeToRetract(s)"
    Label (28,90 150x30), "Mode Selection"
    Rectangle (49,141 314x151)
    Label (30,309 150x30), "bError"
    Lamp1 (126,301 185x47), variable: MAIN.afbPneumaticAxes[MAIN.hmiPneumaticAxisSelection].stPneumaticAxisStruct.stPneumaticAxisStatus.bError, style: Lamp-Lamp1-Red
    Label (37,349 150x30), "E_PneumaticErrors"
    Textfield (169,351 188x30), "%s", text variable: MAIN.afbPneumaticAxes[MAIN.hmiPneumaticAxisSelection].stPneumaticAxisStruct.ePneumaticAxisErrors, text list: 'languageSupport'
    Rectangle (372,256 155x146)
    Rectangle (536,256 158x146)
    Rectangle (372,410 323x181)
    Label (538,259 150x30), "Single Solenoid Manual"
    PushSwitchLed (549,291 50x47), variable: MAIN.afbPneumaticAxes[MAIN.hmiPneumaticAxisSelection].stPneumaticAxisStruct.stPneumaticAxisInputs.bOpenManual, behaviour: TOGGLE, style: Switch-PushSwitchLed-Yellow
    Label (592,293 84x29), "Start Extend"
    Label (557,347 150x30), "Start Retract"
    Label (375,259 150x30), "Single Solenoid PLC"
    PushSwitchLed (387,292 49x49), variable: MAIN.afbPneumaticAxes[MAIN.hmiPneumaticAxisSelection].stPneumaticAxisStruct.stPneumaticAxisControl.bExtend, behaviour: TOGGLE, style: Switch-PushSwitchLed-Yellow
    PushSwitchLed (388,347 48x48), variable: MAIN.afbPneumaticAxes[MAIN.hmiPneumaticAxisSelection].stPneumaticAxisStruct.stPneumaticAxisControl.bRetract, behaviour: TOGGLE, style: Switch-PushSwitchLed-Yellow
    Label (427,418 150x30), "bValveOn"
    Lamp1 (539,419 150x30), variable: MAIN.afbPneumaticAxes[MAIN.hmiPneumaticAxisSelection].stPneumaticAxisStruct.stPneumaticAxisOutputs.bValveOn, style: Lamp-Lamp1-Green
    Label (411,451 150x30), "bMovingExtend"
    Lamp1 (539,451 150x30), variable: MAIN.afbPneumaticAxes[MAIN.hmiPneumaticAxisSelection].stPneumaticAxisStruct.stPneumaticAxisStatus.bExtending, style: Lamp-Lamp1-Green
    Lamp1 (540,483 150x30), variable: MAIN.afbPneumaticAxes[MAIN.hmiPneumaticAxisSelection].stPneumaticAxisStruct.stPneumaticAxisStatus.bRetracting, style: Lamp-Lamp1-Green
    Lamp1 (540,515 150x30), variable: MAIN.afbPneumaticAxes[MAIN.hmiPneumaticAxisSelection].stPneumaticAxisStruct.stPneumaticAxisStatus.bExtended, style: Lamp-Lamp1-Green
    Lamp1 (540,547 150x30), variable: MAIN.afbPneumaticAxes[MAIN.hmiPneumaticAxisSelection].stPneumaticAxisStruct.stPneumaticAxisStatus.bRetracted, style: Lamp-Lamp1-Green
    Label (412,483 150x30), "bMovingRetract"
    Label (426,514 150x30), "bExtended"
    Label (397,294 150x30), "Start Extend"
    Label (398,350 150x30), "Start Retract"
    Label (427,548 150x30), "bRetracted"
    Button (201,304 124x31), "bReset"
        toggle MAIN.afbPneumaticAxes[MAIN.hmiPneumaticAxisSelection].stPneumaticAxisStruct.stPneumaticAxisControl.bReset
    PushSwitchLed (549,346 51x47), variable: MAIN.afbPneumaticAxes[MAIN.hmiPneumaticAxisSelection].stPneumaticAxisStruct.stPneumaticAxisInputs.bCloseManual, behaviour: TOGGLE, style: Switch-PushSwitchLed-Yellow
    Label (84,137 150x30), "bPSSPermit"
    Label (34,222 150x30), "E_PneumaticMode"
    Textfield (165,222 192x30), "%s", text variable: MAIN.afbPneumaticAxes[MAIN.hmiPneumaticAxisSelection].stPneumaticAxisStruct.ePneumaticAxisMode, text list: 'languageSupport'
    Textfield (164,258 192x29), "%s", text variable: MAIN.afbPneumaticAxes[MAIN.hmiPneumaticAxisSelection].stPneumaticAxisStruct.stPneumaticAxisStatus.sStatus, text list: 'languageSupport'
    Label (66,257 150x30), "sStatus"
    Textfield (520,206 82x30), "%d", text variable: MAIN.afbPneumaticAxes[MAIN.hmiPneumaticAxisSelection].stPneumaticAxisStruct.stPneumaticAxisConfig.nTimeToRetract
        OnMouseClick: write MAIN.afbPneumaticAxes[MAIN.hmiPneumaticAxisSelection].stPneumaticAxisStruct.stPneumaticAxisConfig.nTimeToRetract via Default
    Textfield (607,159 75x30), "%d", text variable: MAIN.afbPneumaticAxes[MAIN.hmiPneumaticAxisSelection].fbTimerExtend.ET
    Textfield (608,206 73x30), "%d", text variable: MAIN.afbPneumaticAxes[MAIN.hmiPneumaticAxisSelection].fbTimerRetract.ET
    SpinControl (151,90 207x32), variable: MAIN.afbPneumaticAxes[MAIN.hmiPneumaticAxisSelection].stPneumaticAxisStruct.ePneumaticAxisMode
    Label (570,132 150x30), "Elapsed time (ms)"
    PushSwitchLed (454,77 63x65), variable: MAIN.afbPneumaticAxes[MAIN.hmiPneumaticAxisSelection].stPneumaticAxisStruct.stPneumaticAxisInputs.bEndSwitchBwd, behaviour: TOGGLE, style: Switch-PushSwitchLed-Gray
    PushSwitchLed (543,76 64x65), variable: MAIN.afbPneumaticAxes[MAIN.hmiPneumaticAxisSelection].stPneumaticAxisStruct.stPneumaticAxisInputs.bEndSwitchFwd, behaviour: TOGGLE, style: Switch-PushSwitchLed-Gray
    PushSwitchLed (134,163 53x53), variable: MAIN.afbPneumaticAxes[MAIN.hmiPneumaticAxisSelection].stPneumaticAxisStruct.stPneumaticAxisInputs.bPSSPermit, behaviour: TOGGLE, style: Switch-PushSwitchLed-Gray
    PushSwitchLed (222,164 53x53), variable: MAIN.afbPneumaticAxes[MAIN.hmiPneumaticAxisSelection].stPneumaticAxisStruct.stPneumaticAxisControl.bInterlock, behaviour: TOGGLE, style: Switch-PushSwitchLed-Gray
    Label (171,137 150x30), "bInterlock"
END_VISUALIZATION
